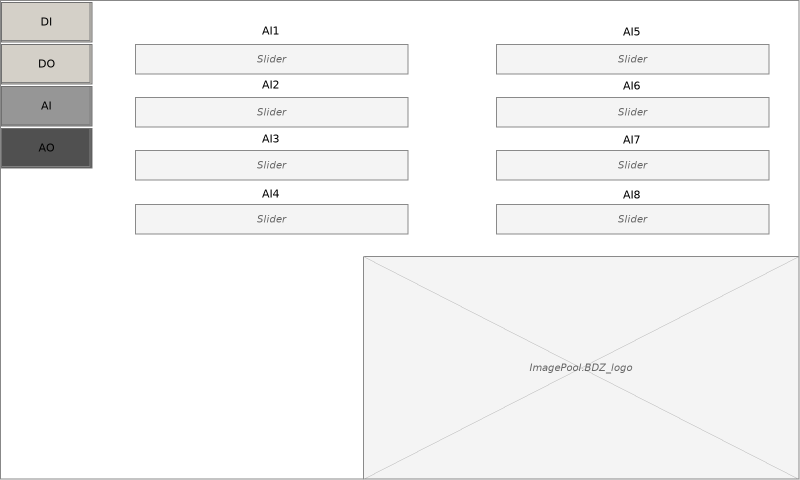
VISUALIZATION Analog_Inputs  // 800x480
    Slider (135,44 273x30), variable: GVL_IO.AI1_ENG, scale 4..20
    Slider (135,97 273x30), variable: GVL_IO.AI2_ENG, scale 4..20
    Slider (135,150 273x30), variable: GVL_IO.AI3_ENG, scale 4..20
    Slider (135,204 273x30), variable: GVL_IO.AI4_ENG, scale 4..20
    Slider (496,44 273x30), variable: GVL_IO.AI5_ENG, scale 4..20
    Slider (496,97 273x30), variable: GVL_IO.AI6_ENG, scale 4..20
    Slider (496,150 273x30), variable: GVL_IO.AI7_ENG, scale 4..20
    Slider (496,204 273x30), variable: GVL_IO.AI8_ENG, scale 4..20
    Label (196,16 150x30), "AI1"
    Label (196,70 150x30), "AI2"
    Label (196,124 150x30), "AI3"
    Label (196,179 150x30), "AI4"
    Label (557,17 150x30), "AI5"
    Label (557,71 150x30), "AI6"
    Label (557,125 150x30), "AI7"
    Label (557,180 150x30), "AI8"
    Button (1,128 91x40), "AO"
        OnMouseUp: change screen: Analog_Outputs
    Button (1,2 91x40), "DI"
        OnMouseUp: change screen: Digital_Inputs
    Button (1,44 91x40), "DO"
        OnMouseDown: change screen: Digital_Outputs
        OnMouseUp: change screen: Digital_Outputs
    Button (1,86 91x40), "AI"
        OnMouseUp: change screen: Analog_Inputs
    Image (363,256 436x223), image: ImagePool.BDZ_logo
END_VISUALIZATION

(* stored: Version 1.1.0.1, ProductVersion 3.1.4024.4
   Visu Analog_Inputs: Id {0f767de4-ae41-46e5-9adb-cd048c3dea72} *)
